Staubli VAL3: PowerOn.pgx

public program PowerOn(bool& x_bBool)
begin
  //
  x_bBool=false
  if workingMode()==4
    if isPowered()==false and esStatus()!=2
      autoConnectMove(true)
      enablePower()
      delay(1)
      x_bBool=true
    endIf
  endIf

end
